Fanuc KAREL source: ko00010.KL

PROGRAM KO00010
%STACKSIZE=65535
%PRIORITY=65535
%NOLOCKGROUP
VAR
P1 : XYZWPR
P2 : XYZWPR
P3 : XYZWPR
OUT : XYZWPR
BEGIN
-- UNRESOLVED_PC line 9 opcodes [27 27 49 7E AD 27 49 7E AD 27 49 7E AD 76 7E 4A] marker_code=0
END KO00010
